FUNCTION_BLOCK StartMotorsTask EXTENDS TcoAbbRoboticsTask



IF Execute() THEN
	 _blink(inOnTime:=T#500MS,inOffTime:=T#500MS);

  	IF _progress = 0 THEN
		IF NOT __ISVALIDREF(inoControl) THEN
			_varInfo :=__VARINFO(inoControl);
			Messenger.Programming(_sb.Clear().Append('<#Invalid reference: #>').Append(_varInfo.Symbol).ToString()).Pin();
		ELSIF NOT __ISVALIDREF(inoConfig) THEN                                                  
			_varInfo :=__VARINFO(inoConfig);                                                    
			Messenger.Programming(_sb.Clear().Append('<#Invalid reference: #>').Append(_varInfo.Symbol).ToString()).Pin();
		ELSIF NOT __ISVALIDREF(inoStatus) THEN                                                  
			_varInfo :=__VARINFO(inoStatus);                                                    
			Messenger.Programming(_sb.Clear().Append('<#Invalid reference: #>').Append(_varInfo.Symbol).ToString()).Pin();
		ELSE

			_progress := _progress + 1;

		END_IF

	END_IF
	IF _progress = 1 THEN
	
		_varInfo :=__VARINFO( inoStatus.State.AutoOn);                                                
		THIS^.Messenger.OnCondition(_infoTimer.Q AND NOT inoStatus.State.AutoOn).Warning(_sb.Clear().Append('<#Waiting for Auto signal! #>').Append(_varInfo.Symbol).ToString());
		IF  inoStatus.State.AutoOn THEN
			_progress := _progress + 1;
		END_IF;
	END_IF;
	
	
	IF _progress = 2 THEN	
		Messenger.Debug('<#Robot Error Reset#>');
		inoControl.ResetError := inoStatus.State.Error AND _blink.outQ;
		IF NOT inoStatus.State.Error THEN
			inoControl.ResetError:=FALSE;
			_progress := _progress + 1;
		END_IF
	END_IF;
	
	IF _progress = 3 THEN	
		Messenger.Debug('<#Robot Emergency Stop Reset#>');
		inoControl.ResetEmgStop := inoStatus.State.EmgStop AND _blink.outQ;
		IF NOT inoStatus.State.EmgStop THEN
			inoControl.ResetEmgStop:=FALSE;
			_progress := _progress + 1;
		END_IF
	END_IF;
		
	
	IF _progress = 4 THEN	
		IF inoStatus.State.Error THEN 
			_progress := 1;
		END_IF
		_varInfo :=__VARINFO( inoStatus.State.MotorOnState);                                                
		THIS^.Messenger.OnCondition(_infoTimer.Q AND NOT inoStatus.State.MotorOnState).Warning(_sb.Clear().Append('<# Waiting for signal: #>').Append(_varInfo.Symbol).ToString());
			_varInfo :=__VARINFO( inoStatus.State.Error);                                                
		THIS^.Messenger.OnCondition(_infoTimer.Q AND NOT inoStatus.State.Error).Warning(_sb.Clear().Append('<# Waiting for signal: #>').Append(_varInfo.Symbol).ToString());
	
		inoControl.MotorOn:=_blink.outQ;	
		IF inoStatus.State.MotorOnState  AND NOT inoStatus.State.Error THEN
			 inoControl.MotorOn:=FALSE;
			_progress := _progress + 1;
		END_IF
	END_IF;		
	
	
	
	
    DoneWhen(inoStatus.State.MotorOnState AND NOT inoStatus.State.Error);
    CallTimers(TRUE);
	
	THIS^.ThrowWhen(_errorTimer.Q or inoStatus.State.Error);
	
END_IF

IF  THIS^.Error AND NOT _errorMessage.Pinned THEN
	THIS^.Restore();
END_IF

METHOD PUBLIC FB_init : BOOL
VAR_INPUT
    bInitRetains : BOOL; // if TRUE, the retain variables are initialized (warm start / cold start)
    bInCopyCode : BOOL; // if TRUE, the instance afterwards gets moved into the copy code (online change)
    ParentObject : ITcoObject;	
END_VAR
END_METHOD

(*~
	<docu>
		<summary>
			Executes when task is aborted.
		</summary>			
	</docu>	
~*)
METHOD PROTECTED OnAbort
IF  __ISVALIDREF(inoStatus) THEN   THIS^.inoStatus.ActionDescription := '<#Start motors  was aborted.#>'; END_IF;
END_METHOD

(*~
	<docu>
		<summary>
			Executes when task reaches the ```Done``` state .
		</summary>			
	</docu>	
~*)
METHOD PROTECTED OnDone
IF  __ISVALIDREF(inoStatus) THEN   THIS^.inoStatus.ActionDescription := '<#Start motors  finished successfully.#>'; END_IF;
_progress:=0;
END_METHOD

METHOD PROTECTED OnError
VAR
	description: STRING;
END_VAR
description := '<#Start motors finished with error.#>'; 
IF  __ISVALIDREF(inoStatus) THEN   THIS^.inoStatus.ActionDescription := description; END_IF;
THIS^._errorMessage.Error(_sb.Clear().Append(description).Append(' To restore acknowledge this alarm.').ToString()).Pin();
END_METHOD

METHOD PROTECTED OnStart
IF  __ISVALIDREF(inoStatus) THEN  THIS^.inoStatus.ActionDescription := '<#Start motors started.#>'; END_IF; 
CallTimers(FALSE);
END_METHOD

(*~
	<docu>
		<summary>
			Restores this instance to the Ready state. Can be called explicitly or from within one of the restore mechanisms.
			<para>
				See also <see cref="PlcDocu.TcoCore.TcoTask.AutoRestorable()"/>
			</para>
		</summary>			
	</docu>	
~*)
METHOD Restore : ITcoRestorable
SUPER^.Restore();
END_METHOD

END_FUNCTION_BLOCK

(* stored: Version 1.1.0.1, ProductVersion 3.1.4024.12
   POU StartMotorsTask: Id {90007edc-04d7-0df9-1d24-a4d6e133c647}, SpecialFunc None
   Method FB_init: Id {063c6942-8f7a-054f-3536-8a61fe16b714}
   Method OnAbort: Id {024284bb-c89c-08e3-2003-dbd51837f544}
   Method OnDone: Id {1d175901-a5df-08b2-35b6-5a962cc9d0c9}
   Method OnError: Id {421042f9-5277-0bc5-31f9-6fec70264897}
   Method OnStart: Id {fcafa02c-1e47-0c37-102f-8c90b5ae05af}
   Method Restore: Id {57998319-88f1-0272-2abe-5f64266a6558} *)
